Staubli VAL3: motionReporter.pgx

program motionReporter()
begin
  while true
    wait(reportEnabled)

    while reportEnabled
      call sendStatus()
      delay(reportInterval)
    endWhile
  endWhile
end
